FUNCTION_BLOCK FB_Shield
VAR_INPUT
END_VAR
VAR_OUTPUT
	Axis_ready					:BOOL:=FALSE;
END_VAR
VAR

ShieldServo: 		FB_AxisControl;

_Shield_param				:recipe;

distance1:					LREAL:=67;




ToolPositioningSpeed	: LREAL := 20;
ToolPositioningAccel	: LREAL := 100;
ToolPositioningJerk		: LREAL := 1000;
ToolHomingSpeed			: LREAL := 2;

ShieldServoEnable:  BOOL;
ShieldServoEnabled: BOOL;

_ExecutedHome				:BOOL:=FALSE;
_ExecutedStage2 			:BOOL:=FALSE;
_ExecutedStage3				:BOOL:=FALSE;
_ExecutedOffset				:BOOL:=FALSE;

tickcounter_shield: 		INT :=0;
State: 						INT:= 0;
StateNext: 					INT:= 0;

END_VAR

METHOD _absolute_move : BOOL
VAR_INPUT
	Enable				:BOOL;
	Stage				:INT;
END_VAR
IF Enable AND NOT Axis_ready THEN
	CASE State OF
	
	0:	
		
		ShieldServo.fPosition:= _Shield_Param.Shield.Distance[Stage];
		ShieldServo.fVelocity:= _Shield_Param.Shield.Speed[Stage]; //mm/s
	
	
		ShieldServo.xMoveA:=TRUE;
	
	
		StateNext:=5;
	5:	
		IF ShieldServo.xInPosition = TRUE THEN
		
			ShieldServo.xMoveA := FALSE;
			StateNext:=0;
			axis_ready:=TRUE;
		
		
		END_IF


	END_CASE

	State:=StateNext;
ELSIF NOT enable THEN
	axis_ready:=FALSE;
	ShieldServo.xMoveA := FALSE;
	state:=0;
END_IF
END_METHOD

METHOD _Enable 
VAR_INPUT
END_VAR

ShieldServoEnable := TRUE;
END_METHOD

METHOD _force_home  : BOOL
VAR_INPUT
	Enable				:BOOL;
	
END_VAR
IF enable AND NOT axis_ready THEN
	CASE State OF
	
	0:	
	
		ShieldServo.fPosition:= 0;
		ShieldServo.fVelocity:= 10; //mm/s
	
		ShieldServo.xMoveA:=TRUE;
		StateNext:=5;
	5:	
		IF ShieldServo.xInPosition = TRUE THEN
		
			ShieldServo.xMoveA := FALSE;
			StateNext:=0;
			axis_ready:=TRUE;
		
		END_IF


	END_CASE

	State:=StateNext;
ELSIF enable = FALSE THEN
	axis_ready:=FALSE;
	ShieldServo.xMoveA := FALSE;
	state:=0;
END_IF
END_METHOD

METHOD _Halt : BOOL
VAR_INPUT
END_VAR
ShieldServo.xHalt:=TRUE;
END_METHOD

METHOD _Halt_false : BOOL
VAR_INPUT
END_VAR
ShieldServo.xHalt:=FALSE;
END_METHOD

METHOD _Home 
VAR_INPUT
	
END_VAR


VAR



END_VAR

VAR_OUTPUT
	
END_VAR





CASE State OF //you are here



0:	
	_ExecutedHome := FALSE;
	ShieldServo.fVelocity := ToolPositioningSpeed;
	ShieldServo.fAxisAcceleration := ToolPositioningAccel;
	ShieldServo.fAxisDeceleration := ToolPositioningAccel;
	ShieldServo.fAxisJerk := ToolPositioningJerk;

	IF ixShieldHomeSwitch THEN
		ShieldServo.xPositiveDirection := FALSE;
		IF  tickcounter_shield < 10 THEN
			tickcounter_shield := tickcounter_shield + 1;  // can be put in onditional
		
		ELSE
		//IF tickcounter_compress >= 10 THEN
			ShieldServo.xMoveV := TRUE;
		END_IF
	ELSE
	
		//CompressServo.xHalt := NOT CompressServo.xHalt;
		ShieldServo.xMoveV := FALSE;
		//CompressServo.xHalt := NOT CompressServo.xHalt;
		ShieldServo.xHalt := TRUE;
		IF ShieldServo.xHalted THEN
			tickcounter_shield:=0;
			StateNext := 5;
		END_IF
	
	END_IF
	
5:
	
	ShieldServo.xHalt := FALSE;
	tickcounter_shield := tickcounter_shield + 1;
	IF tickcounter_shield >= 10 THEN
		tickcounter_shield := 0;
		StateNext := 10;
	END_IF
	
10:
	ShieldServo.fVelocity := ToolHomingSpeed;
	
	IF NOT ixShieldHomeSwitch THEN
		ShieldServo.xPositiveDirection := TRUE;
		IF tickcounter_shield < 10 THEN
			tickcounter_shield := tickcounter_shield + 1;
		ELSE
		//IF tickcounter >= 10 THEN
			shieldServo.xMoveV := TRUE;
		END_IF
	ELSE
		shieldServo.xMoveV := FALSE;
		shieldServo.xHalt := TRUE;
		IF shieldServo.xHalted AND shieldservo.fstandstill THEN
			tickcounter_shield := 0;
			StateNext := 15;
		END_IF
	END_IF

15:
	
	shieldServo.xHalt := FALSE;
	tickcounter_shield := tickcounter_shield + 1;
	IF tickcounter_shield >= 25 THEN
		tickcounter_shield := 0;
		StateNext := 20;
		//Executed := TRUE;
	END_IF
20:
	shieldServo.fHomeOffset := 0;
	shieldServo.xZero := TRUE;
	StateNext := 25;	
	
25:
	IF shieldServo.xZeroed THEN
		shieldServo.xZero := FALSE;
		_ExecutedHome := TRUE;
		StateNext := 0;
	END_IF
	

END_CASE

State := StateNext;
END_METHOD

METHOD _mc_stop : BOOL
VAR_INPUT
END_VAR
ShieldServo.xStop:=TRUE;
END_METHOD

METHOD _Reset
VAR_INPUT
END_VAR
	tickcounter_Shield:=0;
	ShieldServoEnable := FALSE;
	ShieldServo.xZero := FALSE;
	ShieldServo.xMoveV := FALSE;
	ShieldServo.xMoveA := FALSE;
	ShieldServo.xHalt := FALSE;
	ShieldServo.GearIn := FALSE;
	ShieldServo.xStop:=FALSE;
	state:=0;
	statenext:=0;
	
	
	axis_ready:=FALSE;
	_ExecutedHome:=FALSE;
	_ExecutedOffset:=FALSE;
	PRG_Machine.reset_rec_old();
	PRG_Machine._debug(enable:=FALSE);
END_METHOD

METHOD _Reset_medium
VAR_INPUT
END_VAR
	tickcounter_Shield:=0;
	ShieldServoEnable := FALSE;
	ShieldServo.xZero := FALSE;
	ShieldServo.xMoveV := FALSE;
	ShieldServo.xMoveA := FALSE;
	ShieldServo.xHalt := FALSE;
	ShieldServo.GearIn := FALSE;
	ShieldServo.xStop:=FALSE;
	state:=0;
	statenext:=0;
	
	axis_ready:=FALSE;
	PRG_Machine._debug(enable:=FALSE);
END_METHOD

METHOD _retract  : BOOL
VAR_INPUT
	Enable				:BOOL;
	
END_VAR
IF enable AND NOT axis_ready THEN
	CASE State OF
	
	0:	
	
		ShieldServo.fPosition:= 0;
		ShieldServo.fVelocity:= _Shield_Param.Pusher.Retract_Speed; //mm/s
	
		ShieldServo.xMoveA:=TRUE;
		StateNext:=5;
	5:	
		IF ShieldServo.xInPosition = TRUE THEN
		
			ShieldServo.xMoveA := FALSE;
			StateNext:=0;
			axis_ready:=TRUE;
		
		END_IF


	END_CASE

	State:=StateNext;
ELSIF enable = FALSE THEN
	axis_ready:=FALSE;
	ShieldServo.xMoveA := FALSE;
	state:=0;
END_IF
END_METHOD

METHOD _Soft_Reset
VAR_INPUT
END_VAR

tickcounter_Shield:=0;
ShieldServo.xZero := FALSE;
ShieldServo.xMoveV := FALSE;
ShieldServo.xMoveA := FALSE;
ShieldServo.xHalt := FALSE;
ShieldServo.GearIn := FALSE;
ShieldServo.xStop:=FALSE;
state:=0;
statenext:=0;

axis_ready:=FALSE;
PRG_Machine._debug(enable:=FALSE);
END_METHOD

METHOD _Update
VAR_INPUT
END_VAR
ShieldServo(
	xEnable:= ShieldServoEnable, 
	xZero:= , 
	xMoveR:= , 
	xMoveA:= , 
	xMoveV:= , 
	xPositiveDirection:= , 
	fDistance:= , 
	fPosition:= , 
	fVelocity:= , 
	xStop:= , 
	xHome:= , 
	xHomeFlag:= , 
	homePosition:=0,
	fActualPosition=> , 
	fActualVelocity=> , 
	fActModuloPos=> , 
	xEnabled=> ShieldServoEnabled, 
	xMoveComplete=> , 
	xInPosition=> , 
	xAtSpeed=> , 
	xStopped=> , 
	xHomed=> ,
	errorID=> ShieldServoErrorID, 
	Axis:= ShieldAxis );
END_METHOD

PROPERTY HomeExecuted : BOOL;
GET
HomeExecuted := _ExecutedHome;
END_GET
SET
_ExecutedHome := HomeExecuted;
END_SET
END_PROPERTY

METHOD Offset
VAR_INPUT
	Enable				:BOOL;
END_VAR

IF enable AND NOT axis_ready THEN	
	CASE State OF
	0:	
		_ExecutedOffset:=FALSE;
		ShieldServo.fPosition:= _Shield_Param.Other.Shield_Home_Offset-PRG_Machine.rec_old.other.shield_home_offset;
		ShieldServo.fVelocity:= 20; //mm/s
	
		IF ShieldServo.fPosition<>0 THEN
			ShieldServo.xMoveA:=TRUE;
			StateNext:=5;
		ELSE
			_ExecutedOffset:=TRUE;
		END_IF
	
		//StateNext:=5;
	5:	
		IF ShieldServo.xInPosition = TRUE AND ShieldServo.fstandstill THEN
			
			ShieldServo.xMoveA := FALSE;
			StateNext:=7;
			//_ExecutedOffset:=TRUE;
		
		END_IF
		
	7:
		tickcounter_shield:=tickcounter_shield+1;
		IF tickcounter_shield >= 25 THEN
			tickcounter_shield := 0;
			StateNext := 10;
			//Executed := TRUE;
		END_IF
		
	10:
	
		ShieldServo.fHomeOffset := 0;
		ShieldServo.xZero := TRUE;
		StateNext := 15;	
	
	15:
		IF shieldServo.xZeroed THEN
			shieldServo.xZero := FALSE;
			_ExecutedOffset:=TRUE;
			axis_ready:=TRUE;
			StateNext := 0;
		END_IF

	END_CASE

	State:=StateNext;
	
ELSIF NOT enable THEN 
	axis_ready:=FALSE;
	ShieldServo.xZero := FALSE;
	
	StateNext := 0;
END_IF
END_METHOD

PROPERTY OffsetExecuted : BOOL
GET
OffsetExecuted := _ExecutedOffset;
END_GET
SET
_ExecutedOffset := OffsetExecuted;
END_SET
END_PROPERTY

PROPERTY Shield_Param : recipe
GET
Shield_param := _Shield_Param;
END_GET
SET
_Shield_param := Shield_Param;
END_SET
END_PROPERTY

PROPERTY Stage2Executed : BOOL
GET
Stage2Executed := _ExecutedStage2;
END_GET
SET
_ExecutedStage2 := Stage2Executed;
END_SET
END_PROPERTY

PROPERTY Stage3Executed : BOOL
GET
Stage3Executed := _ExecutedStage3;
END_GET
SET
_ExecutedStage3 := Stage3Executed;
END_SET
END_PROPERTY

END_FUNCTION_BLOCK

(* stored: Version 1.1.0.1, ProductVersion 3.1.4020.12
   POU FB_Shield: Id {3352dd00-6753-4b84-9309-30c70609cccf}, SpecialFunc None
   Folder Executed: Id {091ca137-2593-486b-b02a-704598e1bdd6}
   Folder param: Id {2d7a15b3-5509-4c45-a9de-e190bee23ce1}
   Method _absolute_move: Id {812a1d69-4259-448f-9f71-0b18ef866d53}
   Method _Enable: Id {5b595480-7ec2-438c-aed7-aa99c1626b70}
   Method _force_home: Id {da3a4eb7-a6d0-4967-9e09-625b0cedb37e}
   Method _Halt: Id {49e9819d-c096-4f60-a76d-48f1a5f7f93f}
   Method _Halt_false: Id {0196e673-5b67-4dda-b986-f20184d8afe1}
   Method _Home: Id {e3a2bcf1-6b36-4915-aa6d-4a43f630c251}
   Method _mc_stop: Id {a83a92d0-1844-4b66-a7bf-76cd803e9026}
   Method _Reset: Id {cdcb3ac2-204d-4e94-a6da-468cd6a9322e}
   Method _Reset_medium: Id {63d794c2-992d-4538-a5d7-375c66c1638f}
   Method _retract: Id {e2a2f3b0-3dbe-4b15-a792-38be076fb3fc}
   Method _Soft_Reset: Id {2da89526-0ed1-41c7-8028-03a5a355d04c}
   Method _Update: Id {e575f52b-adc7-4530-8dd3-9d372cbc0431}
   Property HomeExecuted: Id {e265ae74-cefc-4e8e-af51-1c93c793b65f}
   Get Get: Id {5460dff2-7a7a-44e9-8cf1-302c6cebcc0d}
   Set Set: Id {bc437082-c97c-4b9c-bdac-5ba8d04a0563}
   Method Offset: Id {ac5cd27c-8097-45c7-959a-7f6c2239b74f}
   Property OffsetExecuted: Id {eaf95a4e-ebfd-4b3c-80b9-edb10c983831}
   Get Get: Id {7f4e8494-e2b8-4426-9e6e-42651934e629}
   Set Set: Id {33d34100-51f5-49b5-bb9c-5ee8757f5808}
   Property Shield_Param: Id {0bbd424d-32c6-47b3-a2f6-d7e425044b71}
   Get Get: Id {3d9f9446-0c62-4054-8023-ae1262e3c1e8}
   Set Set: Id {3d3a29a7-a133-494b-bc4e-a4fb03bfdd07}
   Property Stage2Executed: Id {71ef17c4-0491-4f17-849e-51a7bd7078b5}
   Get Get: Id {09126dbe-83af-467c-9dbf-b9060da89e1e}
   Set Set: Id {8e686e24-281c-43dc-ae92-e63fc2539ecb}
   Property Stage3Executed: Id {83faec63-6689-46ac-93e2-5fe4e09e4bc2}
   Get Get: Id {aeaf94f5-5c99-413d-b13f-5d87d557803d}
   Set Set: Id {27084202-2476-440f-8fff-572e9fa9e0c2} *)
